// TIA Portal V17 export
// export: Created 2023-02-13T11:16:47.4650946Z, ExportSetting WithDefaults, DisplayName Totally Integrated Automation Portal, DisplayVersion V17, DisplayName TIA Portal Openness, DisplayVersion V17, DisplayName TIA Portal Teamcenter Gateway, DisplayVersion V17, DisplayName TIA Portal Version Control Interface, DisplayVersion V17, DisplayName SINAMICS Startdrive Advanced, DisplayVersion V17, DisplayName SINAMICS Startdrive G130, G150, S120, S150, SINAMICS MV, S210, DisplayVersion V17, DisplayName SINAMICS Startdrive G110M, G120, G120C, G120D, G120P, G115D, DisplayVersion V17, DisplayName STEP 7 Professional, DisplayVersion V17, DisplayName STEP 7 Safety, DisplayVersion V17, DisplayName WinCC Professional, DisplayVersion V17
FUNCTION_BLOCK "Homomix"   // FB18, LAD
{ S7_Optimized_Access := 'TRUE' }
VERSION : 0.1
// stored: AutoNumber true, IsIECCheckEnabled false, IsRetainMemResEnabled false, MemoryReserve 100, SetENOAutomatically false, UDAEnableTagReadback false
   VAR_INPUT
      "Level LL" : Bool;
      IN_FBAV_ProWater : Bool;
      IN_FBAV_HW : Bool;
      IN_FBAV_CIP_Tank : Bool;
      IN_FBAV_CIP_Line : Bool;
      IN_FBAV_Outlet : Bool;
      IN_FBAV_Transfer : Bool;
      IN_FBP_Transfer : Bool;
      IN_FBP_Transfer_SP : Real;
      IN_FBP_CIP : Bool;
      IN_FBP_CIP_SP : Real;
      IN_CIP_Enable : Bool;
      IN_CIP_LineOpen : Bool;
      "CIP Pulse" : Bool;
      "CIP Request OK" : Bool;
      "CIP Supply ON" : Bool;
      "CIP In Progress" : Bool;
      "CIP Complete" : Bool;
      IN_Dose_Run : Bool;
      IN_Dose_Held : Bool;
      IN_Dose_Complete : Bool;
      IN_Dose_Valve_Cmd : Bool;
      IN_Dose_Pump_Cmd : Bool;
      IN_Dose_Pump_Sp : Real;
      IN_Dose_LineOK : Bool;
      "ProWater Ready" : Bool;
      "ProWater En" : Bool;
      "HW Ready" : Bool;
      "HW En" : Bool;
      "CIP Busy" : Bool;
      IN_LDT : Date_And_Time;
   END_VAR
   VAR_OUTPUT
      Out_AV_ProWater : Bool;
      Out_AV_HW : Bool;
      Out_AV_CIP_Tank : Bool;
      Out_AV_CIP_Line : Bool;
      Out_AV_Outlet : Bool;
      Out_AV_Transfer : Bool;
      Out_P_Transfer : Bool;
      Out_P_Transfer_SP : Real;
      Out_P_CIP : Bool;
      Out_P_CIP_SP : Real;
      Out_XA : Bool;
      Out_XA_SP : Real;
      Out_Prod_Ready : Bool;
      Out_Tank_Ready : Bool;
      Out_CIP_Tank_Req : Bool;
      Out_CIP_Line_Req : Bool;
      Out_CIP_LineOpen : Bool;
   END_VAR
   VAR
      Cmd : Struct
         Ready_for_Transfer : Bool;
         "CIP Tank" : Bool;
         "CIP Line" : Bool;
         "Agi Mode" : Bool;
         "Agi ON OFF" : Bool;
      END_STRUCT;
   END_VAR
   VAR RETAIN
      Param : Struct
         "CIP Pump SP" : Real := 50.0;
         "Agi SP" : Real := 50.0;
         Dose_HW_SP : Real;
         Dose_ProWater_SP : Real;
         LastDose_HW : Real;
         LastDose_ProWater : Real;
      END_STRUCT;
   END_VAR
   VAR
      State : Struct
         "Tank LL" : Bool;
         "CIP Tank" : Bool;
         "CIP Tank Ena" : Bool;
         "CIP Line" : Bool;
         "CIP Line Ena" : Bool;
         "CIP Return On" : Bool;
         "Dose EN" : Bool;
         ProWater_Inloading : Bool;
         HW_Inloading : Bool;
         Tank_Inloading : Bool;
         "Ready For Transfer" : Bool;
         "Ready For Transfer EN" : Bool;
         Transfer_On_Prog : Bool;
         "CIP Req" : Bool;
      END_STRUCT;
      Dose : Struct
         Dose_Start : DWord;
         Dose_Pause : DWord;
         Dose_Stop : DWord;
         Dose_State : DWord;
         Dose_Tank_Available : Word;
         Dose_Prod_Ready : Word;
         Dose_Header_Req : DWord;
         Dose_EN : Word;
      END_STRUCT;
      SP_ProWater : "Raw_Pulse";
      SP_HW { S7_SetPoint := 'True'} : "Raw_Pulse";
      Dose_ProWater { S7_SetPoint := 'True'} : "DOSE";
      Dose_HW { S7_SetPoint := 'True'} : "DOSE";
      r : Struct
         PosE1 : Bool;
         PosE2 : Bool;
         PosE3 : Bool;
         PosE4 : Bool;
         PosE5 : Bool;
         PosE6 : Bool;
         PosE7 : Bool;
         PosE8 : Bool;
         PosE9 : Bool;
         PosE10 : Bool;
         PosE11 : Bool;
         PosE12 : Bool;
         PosE13 : Bool;
         PosE14 : Bool;
         PosE15 : Bool;
         PosE16 : Bool;
         PosE17 : Bool;
         PosE18 : Bool;
         PosE19 : Bool;
         PosE20 : Bool;
         PosE21 : Bool;
         PosE22 : Bool;
         PosE23 : Bool;
         PosE24 : Bool;
         PosE25 : Bool;
         PosE26 : Bool;
         PosE27 : Bool;
         PosE28 : Bool;
         PosE29 : Bool;
         PosE30 : Bool;
         PosE31 : Bool;
         PosE32 : Bool;
      END_STRUCT;
      CIPRetOn_Time : TON_TIME;
      CIPRetOff_Time { S7_SetPoint := 'True'} : TON_TIME;
      Actuator : Struct
         AV_Transfer : Bool;
         AV_Outlet : Bool;
         AV_CIP : Bool;
         P_Transfer : Bool;
         P_CIP : Bool;
      END_STRUCT;
      alwaysOn : Bool;
   END_VAR
   VAR RETAIN
      TimerON : Struct
         TimerON_1 : TON_TIME;
         TimerON_2 { S7_SetPoint := 'True'} : TON_TIME;
         TimerON_3 { S7_SetPoint := 'True'} : TON_TIME;
         TimerON_4 { S7_SetPoint := 'True'} : TON_TIME;
         TimerON_5 { S7_SetPoint := 'True'} : TON_TIME;
         TimerON_6 { S7_SetPoint := 'True'} : TON_TIME;
         TimerON_7 { S7_SetPoint := 'True'} : TON_TIME;
         TimerON_8 { S7_SetPoint := 'True'} : TON_TIME;
      END_STRUCT;
   END_VAR
   VAR_TEMP
      b_transfer : Bool;
   END_VAR
   // SP_ProWater.Para."SP_Qty_Fine%" := 10.0;
   // SP_HW.Para."SP_Qty_Fine%" := 10.0;
   // TimerON.TimerON_1.PT := T#10s;
   // TimerON.TimerON_2.PT := T#10s;
   // TimerON.TimerON_3.PT := T#10s;
   // TimerON.TimerON_4.PT := T#10s;
   // TimerON.TimerON_5.PT := T#10s;
   // TimerON.TimerON_6.PT := T#10s;
   // TimerON.TimerON_7.PT := T#10s;
   // TimerON.TimerON_8.PT := T#10s;
   VAR_TEMP   // added for the SCL form of the ladder/FBD networks
      _w1 : Bool;
      _w2 : Bool;
   END_VAR
BEGIN

REGION Network 1: Always ON
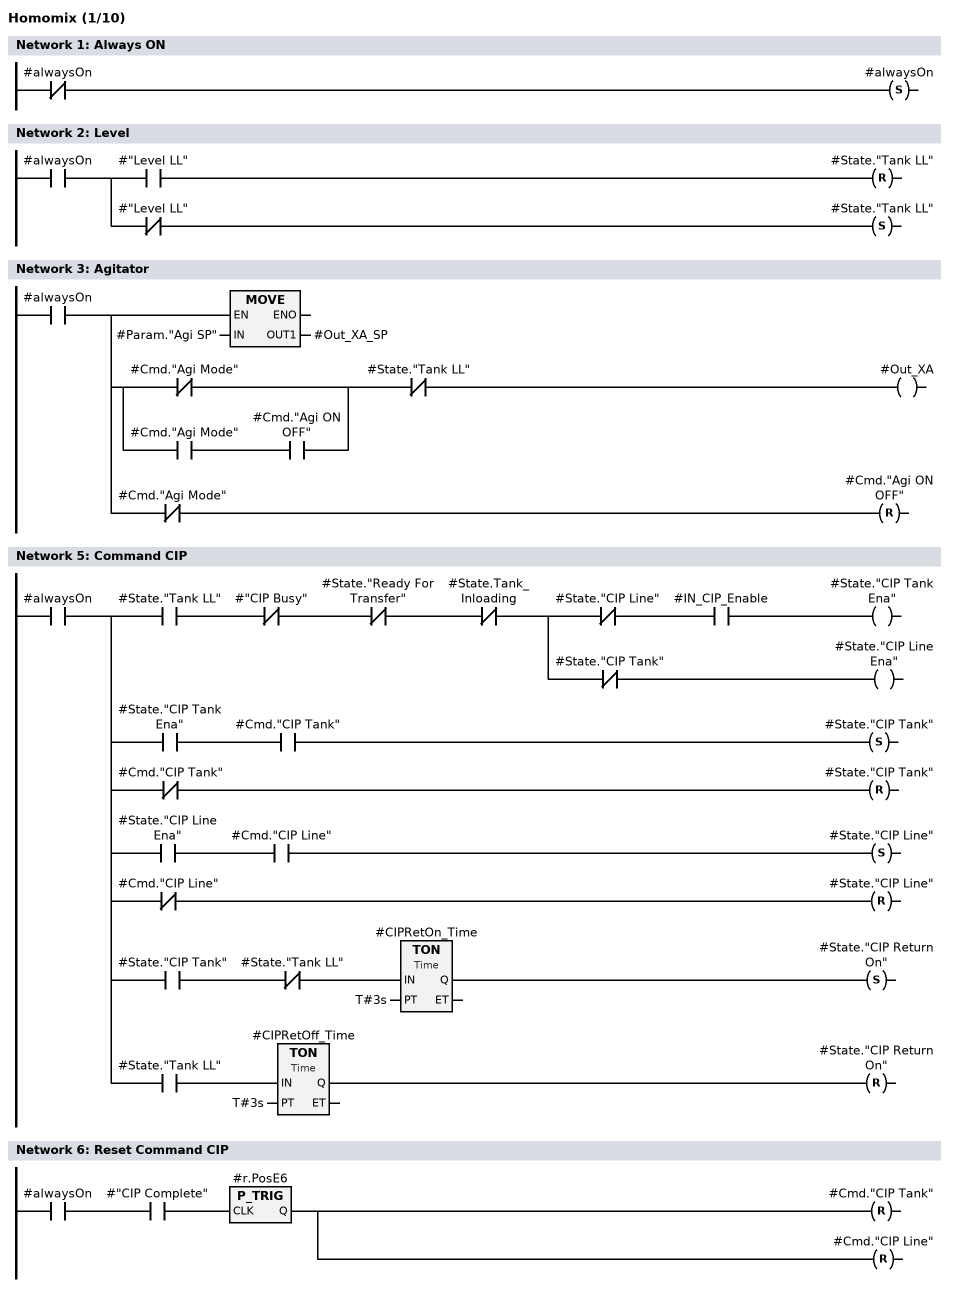
   RUNG wire#powerrail
      I_Contact( #alwaysOn )
      S_Coil( #alwaysOn )
   END_RUNG
   // the same network as SCL:
   IF NOT #alwaysOn THEN #alwaysOn := TRUE; END_IF;
END_REGION

REGION Network 2: Level
   RUNG wire#powerrail
      Contact( #alwaysOn )
      wire#w1
      Contact( #"Level LL" )
      R_Coil( #State."Tank LL" )
   END_RUNG
   RUNG wire#w1
      I_Contact( #"Level LL" )
      S_Coil( #State."Tank LL" )
   END_RUNG
   // the same network as SCL:
   IF #alwaysOn AND #"Level LL" THEN #State."Tank LL" := FALSE; END_IF;
   IF #alwaysOn AND NOT #"Level LL" THEN #State."Tank LL" := TRUE; END_IF;
END_REGION

REGION Network 3: Agitator
   RUNG wire#powerrail
      Contact( #alwaysOn )
      wire#w1
      Move(in := #Param."Agi SP", out1 => #Out_XA_SP)
   END_RUNG
   RUNG wire#w1
      I_Contact( #Cmd."Agi Mode" )
      wire#w2
      I_Contact( #State."Tank LL" )
      Coil( #Out_XA )
   END_RUNG
   RUNG wire#w1
      Contact( #Cmd."Agi Mode" )
      Contact( #Cmd."Agi ON OFF" )
   END_RUNG wire#w2
   RUNG wire#w1
      I_Contact( #Cmd."Agi Mode" )
      R_Coil( #Cmd."Agi ON OFF" )
   END_RUNG
   // the same network as SCL:
   IF #alwaysOn THEN #Out_XA_SP := #Param."Agi SP"; END_IF;
   #Out_XA := #alwaysOn AND (NOT #Cmd."Agi Mode" OR (#Cmd."Agi Mode" AND #Cmd."Agi ON OFF")) AND NOT #State."Tank LL";
   IF #alwaysOn AND NOT #Cmd."Agi Mode" THEN #Cmd."Agi ON OFF" := FALSE; END_IF;
END_REGION

REGION Network 5: Command CIP
   RUNG wire#powerrail
      Contact( #alwaysOn )
      wire#w1
      Contact( #State."Tank LL" )
      I_Contact( #"CIP Busy" )
      I_Contact( #State."Ready For Transfer" )
      I_Contact( #State.Tank_Inloading )
      wire#w2
      I_Contact( #State."CIP Line" )
      Contact( #IN_CIP_Enable )
      Coil( #State."CIP Tank Ena" )
   END_RUNG
   RUNG wire#w2
      I_Contact( #State."CIP Tank" )
      Coil( #State."CIP Line Ena" )
   END_RUNG
   RUNG wire#w1
      Contact( #State."CIP Tank Ena" )
      Contact( #Cmd."CIP Tank" )
      S_Coil( #State."CIP Tank" )
   END_RUNG
   RUNG wire#w1
      I_Contact( #Cmd."CIP Tank" )
      R_Coil( #State."CIP Tank" )
   END_RUNG
   RUNG wire#w1
      Contact( #State."CIP Line Ena" )
      Contact( #Cmd."CIP Line" )
      S_Coil( #State."CIP Line" )
   END_RUNG
   RUNG wire#w1
      I_Contact( #Cmd."CIP Line" )
      R_Coil( #State."CIP Line" )
   END_RUNG
   RUNG wire#w1
      Contact( #State."CIP Tank" )
      I_Contact( #State."Tank LL" )
      { S7_Templates := "time_type := Time" } #CIPRetOn_Time.TON(pt := T#3s, et =>)
      S_Coil( #State."CIP Return On" )
   END_RUNG
   RUNG wire#w1
      Contact( #State."Tank LL" )
      { S7_Templates := "time_type := Time" } #CIPRetOff_Time.TON(pt := T#3s, et =>)
      R_Coil( #State."CIP Return On" )
   END_RUNG
   // the same network as SCL:
   #_w1 := #alwaysOn AND #State."Tank LL" AND NOT #"CIP Busy" AND NOT #State."Ready For Transfer" AND NOT #State.Tank_Inloading;
   #State."CIP Tank Ena" := #_w1 AND NOT #State."CIP Line" AND #IN_CIP_Enable;
   #State."CIP Line Ena" := #_w1 AND NOT #State."CIP Tank";
   IF #alwaysOn AND #State."CIP Tank Ena" AND #Cmd."CIP Tank" THEN #State."CIP Tank" := TRUE; END_IF;
   IF #alwaysOn AND NOT #Cmd."CIP Tank" THEN #State."CIP Tank" := FALSE; END_IF;
   IF #alwaysOn AND #State."CIP Line Ena" AND #Cmd."CIP Line" THEN #State."CIP Line" := TRUE; END_IF;
   IF #alwaysOn AND NOT #Cmd."CIP Line" THEN #State."CIP Line" := FALSE; END_IF;
   #CIPRetOn_Time(IN := #alwaysOn AND #State."CIP Tank" AND NOT #State."Tank LL", PT := T#3s);   // TON
   IF #CIPRetOn_Time.Q THEN #State."CIP Return On" := TRUE; END_IF;
   #CIPRetOff_Time(IN := #alwaysOn AND #State."Tank LL", PT := T#3s);   // TON
   IF #CIPRetOff_Time.Q THEN #State."CIP Return On" := FALSE; END_IF;
END_REGION

REGION Network 6: Reset Command CIP
   RUNG wire#powerrail
      Contact( #alwaysOn )
      Contact( #"CIP Complete" )
      P_Trig( #r.PosE6 )
      wire#w1
      R_Coil( #Cmd."CIP Tank" )
   END_RUNG
   RUNG wire#w1
      R_Coil( #Cmd."CIP Line" )
   END_RUNG
   // the same network as SCL:
   #_w1 := #alwaysOn AND #"CIP Complete";
   #_w2 := #_w1 AND NOT #r.PosE6;   // rising edge
   #r.PosE6 := #_w1;
   IF #_w2 THEN
       #Cmd."CIP Tank" := FALSE;
       #Cmd."CIP Line" := FALSE;
   END_IF;
END_REGION

REGION Network 7: CIP Request and CIP Line Open
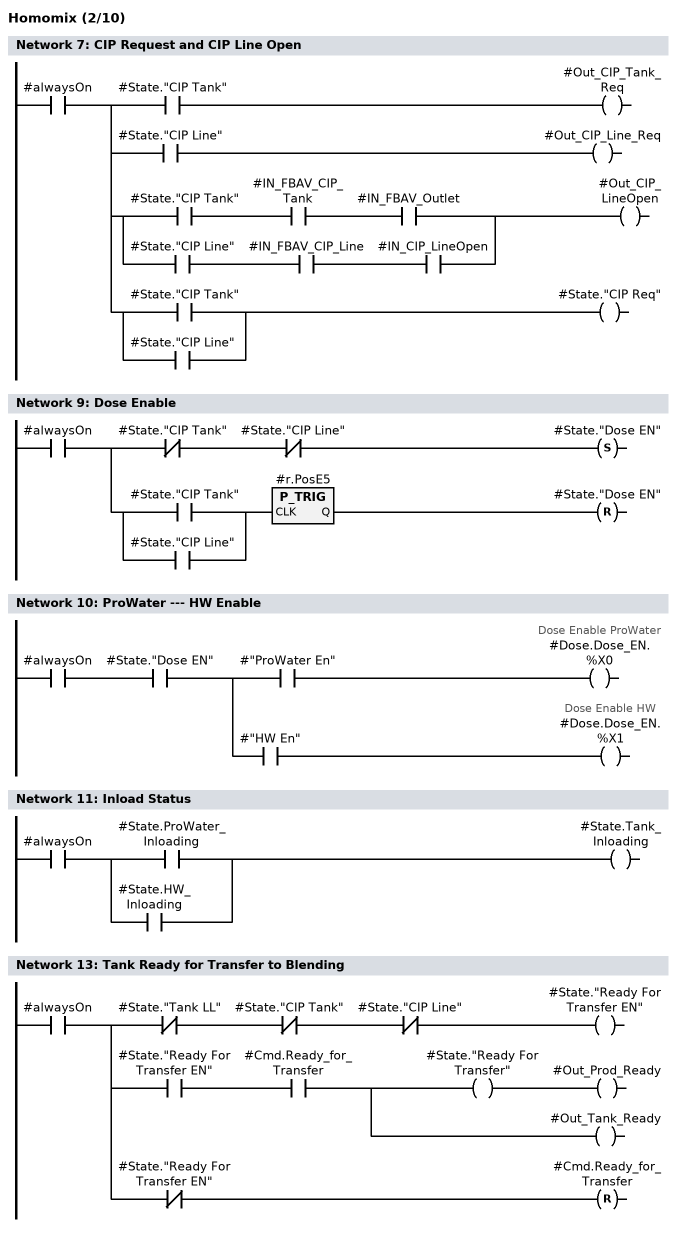
   RUNG wire#powerrail
      Contact( #alwaysOn )
      wire#w1
      Contact( #State."CIP Tank" )
      Coil( #Out_CIP_Tank_Req )
   END_RUNG
   RUNG wire#w1
      Contact( #State."CIP Line" )
      Coil( #Out_CIP_Line_Req )
   END_RUNG
   RUNG wire#w1
      Contact( #State."CIP Tank" )
      Contact( #IN_FBAV_CIP_Tank )
      Contact( #IN_FBAV_Outlet )
      wire#w2
      Coil( #Out_CIP_LineOpen )
   END_RUNG
   RUNG wire#w1
      Contact( #State."CIP Line" )
      Contact( #IN_FBAV_CIP_Line )
      Contact( #IN_CIP_LineOpen )
   END_RUNG wire#w2
   RUNG wire#w1
      Contact( #State."CIP Tank" )
      wire#w3
      Coil( #State."CIP Req" )
   END_RUNG
   RUNG wire#w1
      Contact( #State."CIP Line" )
   END_RUNG wire#w3
   // the same network as SCL:
   #Out_CIP_Tank_Req := #alwaysOn AND #State."CIP Tank";
   #Out_CIP_Line_Req := #alwaysOn AND #State."CIP Line";
   #Out_CIP_LineOpen := #alwaysOn AND ((#State."CIP Tank" AND #IN_FBAV_CIP_Tank AND #IN_FBAV_Outlet) OR (#State."CIP Line" AND #IN_FBAV_CIP_Line AND #IN_CIP_LineOpen));
   #State."CIP Req" := #alwaysOn AND (#State."CIP Tank" OR #State."CIP Line");
END_REGION

REGION Network 9: Dose Enable
   RUNG wire#powerrail
      Contact( #alwaysOn )
      wire#w1
      I_Contact( #State."CIP Tank" )
      I_Contact( #State."CIP Line" )
      S_Coil( #State."Dose EN" )
   END_RUNG
   RUNG wire#w1
      Contact( #State."CIP Tank" )
      wire#w2
      P_Trig( #r.PosE5 )
      R_Coil( #State."Dose EN" )
   END_RUNG
   RUNG wire#w1
      Contact( #State."CIP Line" )
   END_RUNG wire#w2
   // the same network as SCL:
   IF #alwaysOn AND NOT #State."CIP Tank" AND NOT #State."CIP Line" THEN #State."Dose EN" := TRUE; END_IF;
   #_w1 := #alwaysOn AND (#State."CIP Tank" OR #State."CIP Line");
   #_w2 := #_w1 AND NOT #r.PosE5;   // rising edge
   #r.PosE5 := #_w1;
   IF #_w2 THEN #State."Dose EN" := FALSE; END_IF;
END_REGION

REGION Network 10: ProWater --- HW Enable
   RUNG wire#powerrail
      Contact( #alwaysOn )
      Contact( #State."Dose EN" )
      wire#w1
      Contact( #"ProWater En" )
      Coil( #Dose.Dose_EN.%X0 )   // Dose Enable ProWater
   END_RUNG
   RUNG wire#w1
      Contact( #"HW En" )
      Coil( #Dose.Dose_EN.%X1 )   // Dose Enable HW
   END_RUNG
   // the same network as SCL:
   #_w1 := #alwaysOn AND #State."Dose EN";
   #Dose.Dose_EN.%X0 := #_w1 AND #"ProWater En";   // Dose Enable ProWater
   #Dose.Dose_EN.%X1 := #_w1 AND #"HW En";   // Dose Enable HW
END_REGION

REGION Network 11: Inload Status
   RUNG wire#powerrail
      Contact( #alwaysOn )
      wire#w1
      Contact( #State.ProWater_Inloading )
      wire#w2
      Coil( #State.Tank_Inloading )
   END_RUNG
   RUNG wire#w1
      Contact( #State.HW_Inloading )
   END_RUNG wire#w2
   // the same network as SCL:
   #State.Tank_Inloading := #alwaysOn AND (#State.ProWater_Inloading OR #State.HW_Inloading);
END_REGION

REGION Network 13: Tank Ready for Transfer to Blending
   RUNG wire#powerrail
      Contact( #alwaysOn )
      wire#w1
      I_Contact( #State."Tank LL" )
      I_Contact( #State."CIP Tank" )
      I_Contact( #State."CIP Line" )
      Coil( #State."Ready For Transfer EN" )
   END_RUNG
   RUNG wire#w1
      Contact( #State."Ready For Transfer EN" )
      Contact( #Cmd.Ready_for_Transfer )
      wire#w2
      Coil( #State."Ready For Transfer" )
      Coil( #Out_Prod_Ready )
   END_RUNG
   RUNG wire#w2
      Coil( #Out_Tank_Ready )
   END_RUNG
   RUNG wire#w1
      I_Contact( #State."Ready For Transfer EN" )
      R_Coil( #Cmd.Ready_for_Transfer )
   END_RUNG
   // the same network as SCL:
   #State."Ready For Transfer EN" := #alwaysOn AND NOT #State."Tank LL" AND NOT #State."CIP Tank" AND NOT #State."CIP Line";
   #State."Ready For Transfer" := #alwaysOn AND #State."Ready For Transfer EN" AND #Cmd.Ready_for_Transfer;
   #Out_Prod_Ready := #State."Ready For Transfer";
   #Out_Tank_Ready := #State."Ready For Transfer";
   IF #alwaysOn AND NOT #State."Ready For Transfer EN" THEN #Cmd.Ready_for_Transfer := FALSE; END_IF;
END_REGION

REGION Network 14: Transfer to Blending AV and Pump
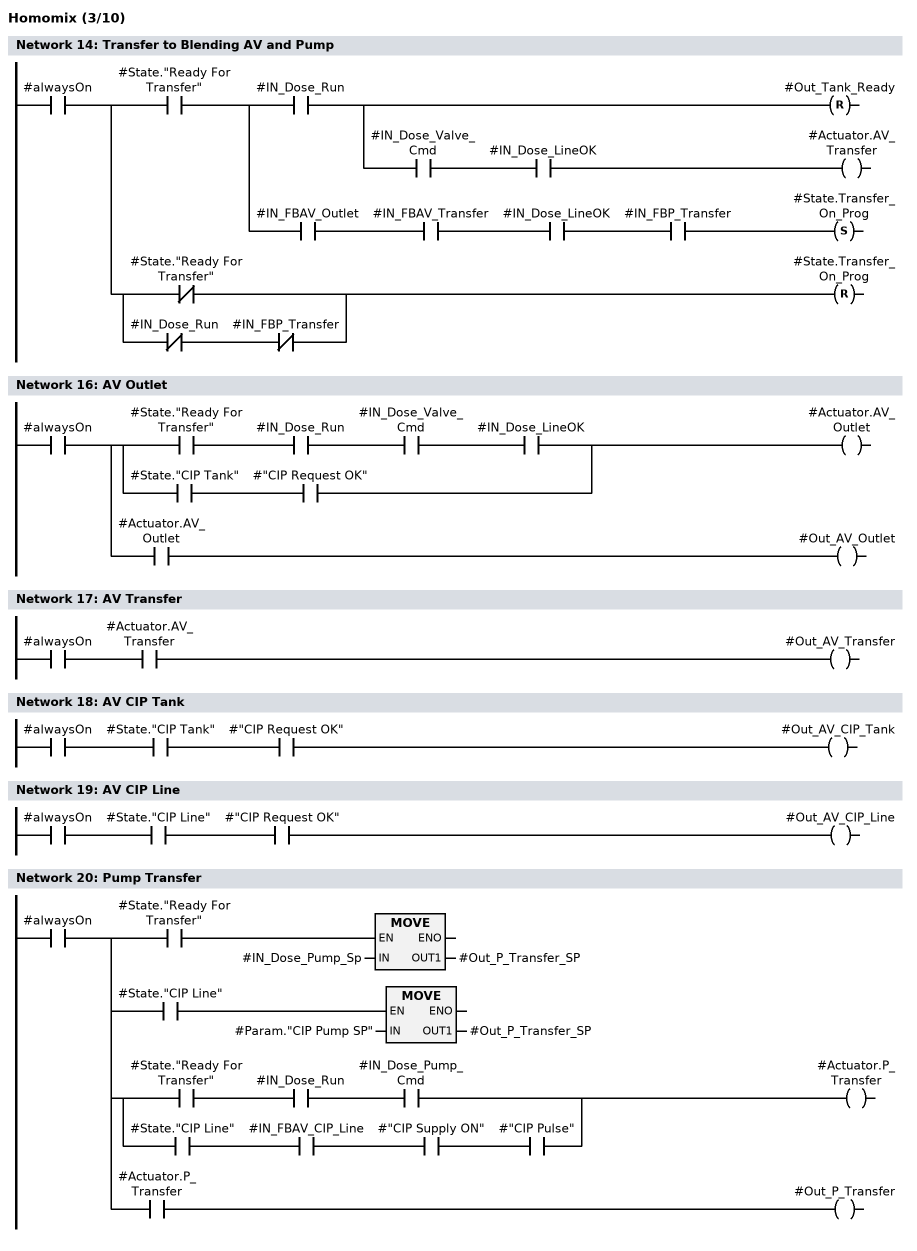
   RUNG wire#powerrail
      Contact( #alwaysOn )
      wire#w1
      Contact( #State."Ready For Transfer" )
      wire#w2
      Contact( #IN_Dose_Run )
      wire#w3
      R_Coil( #Out_Tank_Ready )
   END_RUNG
   RUNG wire#w3
      Contact( #IN_Dose_Valve_Cmd )
      Contact( #IN_Dose_LineOK )
      Coil( #Actuator.AV_Transfer )
   END_RUNG
   RUNG wire#w2
      Contact( #IN_FBAV_Outlet )
      Contact( #IN_FBAV_Transfer )
      Contact( #IN_Dose_LineOK )
      Contact( #IN_FBP_Transfer )
      S_Coil( #State.Transfer_On_Prog )
   END_RUNG
   RUNG wire#w1
      I_Contact( #State."Ready For Transfer" )
      wire#w4
      R_Coil( #State.Transfer_On_Prog )
   END_RUNG
   RUNG wire#w1
      I_Contact( #IN_Dose_Run )
      I_Contact( #IN_FBP_Transfer )
   END_RUNG wire#w4
   // the same network as SCL:
   #_w1 := #alwaysOn AND #State."Ready For Transfer";
   #_w2 := #_w1 AND #IN_Dose_Run;
   IF #_w2 THEN #Out_Tank_Ready := FALSE; END_IF;
   #Actuator.AV_Transfer := #_w2 AND #IN_Dose_Valve_Cmd AND #IN_Dose_LineOK;
   IF #_w1 AND #IN_FBAV_Outlet AND #IN_FBAV_Transfer AND #IN_Dose_LineOK AND #IN_FBP_Transfer THEN
       #State.Transfer_On_Prog := TRUE;
   END_IF;
   IF #alwaysOn AND (NOT #State."Ready For Transfer" OR (NOT #IN_Dose_Run AND NOT #IN_FBP_Transfer)) THEN
       #State.Transfer_On_Prog := FALSE;
   END_IF;
END_REGION

REGION Network 16: AV Outlet
   RUNG wire#powerrail
      Contact( #alwaysOn )
      wire#w1
      Contact( #State."Ready For Transfer" )
      Contact( #IN_Dose_Run )
      Contact( #IN_Dose_Valve_Cmd )
      Contact( #IN_Dose_LineOK )
      wire#w2
      Coil( #Actuator.AV_Outlet )
   END_RUNG
   RUNG wire#w1
      Contact( #State."CIP Tank" )
      Contact( #"CIP Request OK" )
   END_RUNG wire#w2
   RUNG wire#w1
      Contact( #Actuator.AV_Outlet )
      Coil( #Out_AV_Outlet )
   END_RUNG
   // the same network as SCL:
   #Actuator.AV_Outlet := #alwaysOn AND ((#State."Ready For Transfer" AND #IN_Dose_Run AND #IN_Dose_Valve_Cmd AND #IN_Dose_LineOK) OR (#State."CIP Tank" AND #"CIP Request OK"));
   #Out_AV_Outlet := #alwaysOn AND #Actuator.AV_Outlet;
END_REGION

REGION Network 17: AV Transfer
   RUNG wire#powerrail
      Contact( #alwaysOn )
      Contact( #Actuator.AV_Transfer )
      Coil( #Out_AV_Transfer )
   END_RUNG
   // the same network as SCL:
   #Out_AV_Transfer := #alwaysOn AND #Actuator.AV_Transfer;
END_REGION

REGION Network 18: AV CIP Tank
   RUNG wire#powerrail
      Contact( #alwaysOn )
      Contact( #State."CIP Tank" )
      Contact( #"CIP Request OK" )
      Coil( #Out_AV_CIP_Tank )
   END_RUNG
   // the same network as SCL:
   #Out_AV_CIP_Tank := #alwaysOn AND #State."CIP Tank" AND #"CIP Request OK";
END_REGION

REGION Network 19: AV CIP Line
   RUNG wire#powerrail
      Contact( #alwaysOn )
      Contact( #State."CIP Line" )
      Contact( #"CIP Request OK" )
      Coil( #Out_AV_CIP_Line )
   END_RUNG
   // the same network as SCL:
   #Out_AV_CIP_Line := #alwaysOn AND #State."CIP Line" AND #"CIP Request OK";
END_REGION

REGION Network 20: Pump Transfer
   RUNG wire#powerrail
      Contact( #alwaysOn )
      wire#w1
      Contact( #State."Ready For Transfer" )
      Move(in := #IN_Dose_Pump_Sp, out1 => #Out_P_Transfer_SP)
   END_RUNG
   RUNG wire#w1
      Contact( #State."CIP Line" )
      Move(in := #Param."CIP Pump SP", out1 => #Out_P_Transfer_SP)
   END_RUNG
   RUNG wire#w1
      Contact( #State."Ready For Transfer" )
      Contact( #IN_Dose_Run )
      Contact( #IN_Dose_Pump_Cmd )
      wire#w2
      Coil( #Actuator.P_Transfer )
   END_RUNG
   RUNG wire#w1
      Contact( #State."CIP Line" )
      Contact( #IN_FBAV_CIP_Line )
      Contact( #"CIP Supply ON" )
      Contact( #"CIP Pulse" )
   END_RUNG wire#w2
   RUNG wire#w1
      Contact( #Actuator.P_Transfer )
      Coil( #Out_P_Transfer )
   END_RUNG
   // the same network as SCL:
   IF #alwaysOn AND #State."Ready For Transfer" THEN #Out_P_Transfer_SP := #IN_Dose_Pump_Sp; END_IF;
   IF #alwaysOn AND #State."CIP Line" THEN #Out_P_Transfer_SP := #Param."CIP Pump SP"; END_IF;
   #Actuator.P_Transfer := #alwaysOn AND ((#State."Ready For Transfer" AND #IN_Dose_Run AND #IN_Dose_Pump_Cmd) OR (#State."CIP Line" AND #IN_FBAV_CIP_Line AND #"CIP Supply ON" AND #"CIP Pulse"));
   #Out_P_Transfer := #alwaysOn AND #Actuator.P_Transfer;
END_REGION

REGION Network 21: Pump CIP Tank
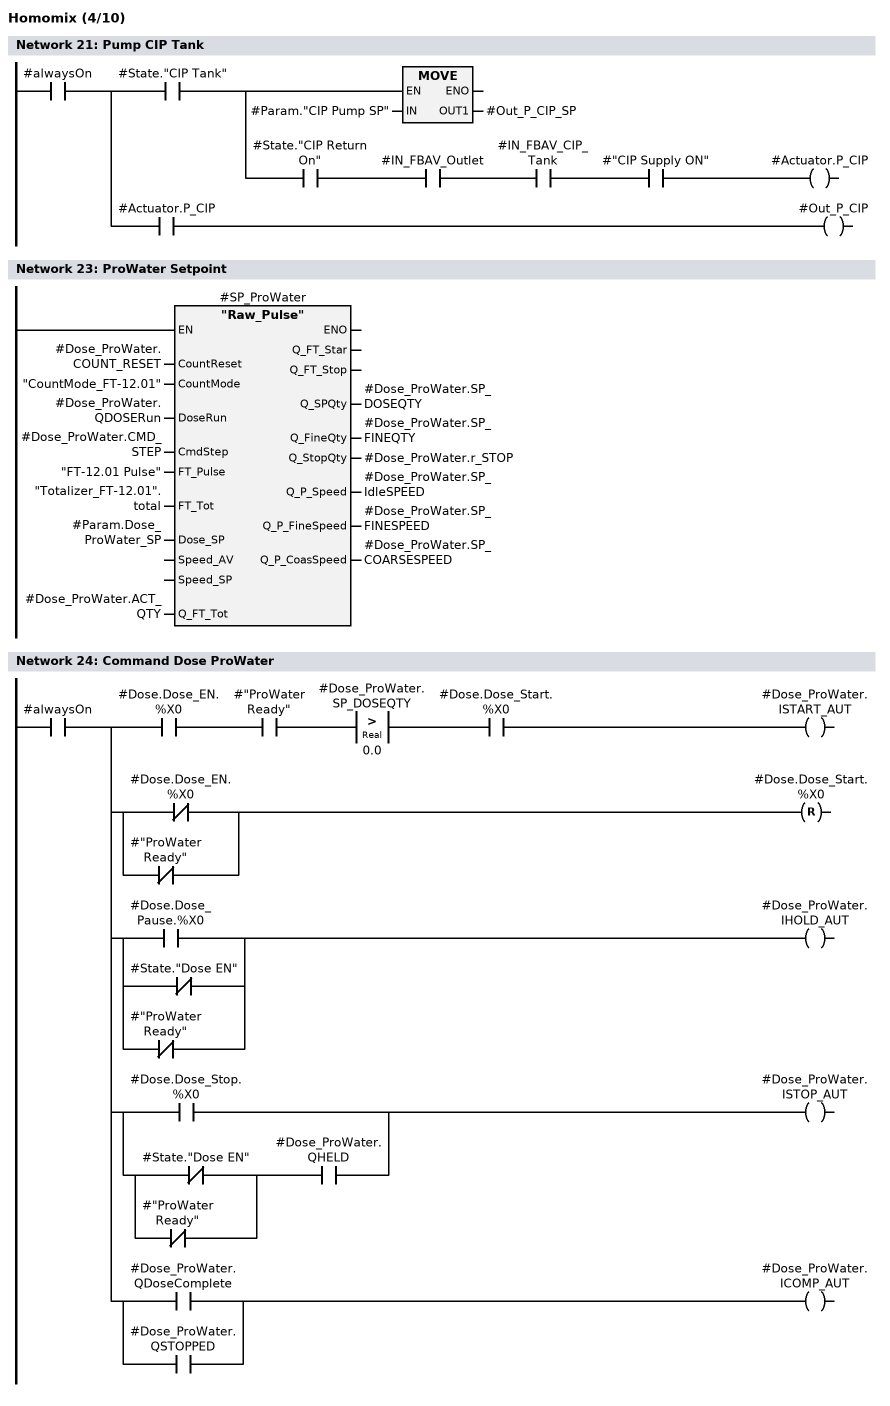
   RUNG wire#powerrail
      Contact( #alwaysOn )
      wire#w1
      Contact( #State."CIP Tank" )
      wire#w2
      Move(in := #Param."CIP Pump SP", out1 => #Out_P_CIP_SP)
   END_RUNG
   RUNG wire#w2
      Contact( #State."CIP Return On" )
      Contact( #IN_FBAV_Outlet )
      Contact( #IN_FBAV_CIP_Tank )
      Contact( #"CIP Supply ON" )
      Coil( #Actuator.P_CIP )
   END_RUNG
   RUNG wire#w1
      Contact( #Actuator.P_CIP )
      Coil( #Out_P_CIP )
   END_RUNG
   // the same network as SCL:
   #_w1 := #alwaysOn AND #State."CIP Tank";
   IF #_w1 THEN #Out_P_CIP_SP := #Param."CIP Pump SP"; END_IF;
   #Actuator.P_CIP := #_w1 AND #State."CIP Return On" AND #IN_FBAV_Outlet AND #IN_FBAV_CIP_Tank AND #"CIP Supply ON";
   #Out_P_CIP := #alwaysOn AND #Actuator.P_CIP;
END_REGION

REGION Network 23: ProWater Setpoint
   RUNG wire#powerrail
      #SP_ProWater(CountReset := #Dose_ProWater.COUNT_RESET, CountMode := "CountMode_FT-12.01", DoseRun := #Dose_ProWater.QDOSERun, CmdStep := #Dose_ProWater.CMD_STEP, FT_Pulse := "FT-12.01 Pulse", FT_Tot := "Totalizer_FT-12.01".total, Dose_SP := #Param.Dose_ProWater_SP, Speed_AV :=, Speed_SP :=, Q_FT_Tot := #Dose_ProWater.ACT_QTY, Q_FT_Star =>, Q_FT_Stop =>, Q_SPQty => #Dose_ProWater.SP_DOSEQTY, Q_FineQty => #Dose_ProWater.SP_FINEQTY, Q_StopQty => #Dose_ProWater.r_STOP, Q_P_Speed => #Dose_ProWater.SP_IdleSPEED, Q_P_FineSpeed => #Dose_ProWater.SP_FINESPEED, Q_P_CoasSpeed => #Dose_ProWater.SP_COARSESPEED)
   END_RUNG
   // the same network as SCL:
   #SP_ProWater(CountReset := #Dose_ProWater.COUNT_RESET,   // "Raw_Pulse"
                CountMode := "CountMode_FT-12.01",
                DoseRun := #Dose_ProWater.QDOSERun,
                CmdStep := #Dose_ProWater.CMD_STEP,
                FT_Pulse := "FT-12.01 Pulse",
                FT_Tot := "Totalizer_FT-12.01".total,
                Dose_SP := #Param.Dose_ProWater_SP,
                Q_FT_Tot := #Dose_ProWater.ACT_QTY,
                Q_SPQty => #Dose_ProWater.SP_DOSEQTY,
                Q_FineQty => #Dose_ProWater.SP_FINEQTY,
                Q_StopQty => #Dose_ProWater.r_STOP,
                Q_P_Speed => #Dose_ProWater.SP_IdleSPEED,
                Q_P_FineSpeed => #Dose_ProWater.SP_FINESPEED,
                Q_P_CoasSpeed => #Dose_ProWater.SP_COARSESPEED);
END_REGION

REGION Network 24: Command Dose ProWater
   RUNG wire#powerrail
      Contact( #alwaysOn )
      wire#w1
      Contact( #Dose.Dose_EN.%X0 )
      Contact( #"ProWater Ready" )
      { S7_Templates := "SrcType := Real" } GT_Contact(in1 := #Dose_ProWater.SP_DOSEQTY, in2 := 0.0)
      Contact( #Dose.Dose_Start.%X0 )
      Coil( #Dose_ProWater.ISTART_AUT )
   END_RUNG
   RUNG wire#w1
      I_Contact( #Dose.Dose_EN.%X0 )
      wire#w2
      R_Coil( #Dose.Dose_Start.%X0 )
   END_RUNG
   RUNG wire#w1
      I_Contact( #"ProWater Ready" )
   END_RUNG wire#w2
   RUNG wire#w1
      Contact( #Dose.Dose_Pause.%X0 )
      wire#w3
      Coil( #Dose_ProWater.IHOLD_AUT )
   END_RUNG
   RUNG wire#w1
      I_Contact( #State."Dose EN" )
   END_RUNG wire#w3
   RUNG wire#w1
      I_Contact( #"ProWater Ready" )
   END_RUNG wire#w3
   RUNG wire#w1
      Contact( #Dose.Dose_Stop.%X0 )
      wire#w4
      Coil( #Dose_ProWater.ISTOP_AUT )
   END_RUNG
   RUNG wire#w1
      I_Contact( #State."Dose EN" )
      wire#w5
      Contact( #Dose_ProWater.QHELD )
   END_RUNG wire#w4
   RUNG wire#w1
      I_Contact( #"ProWater Ready" )
   END_RUNG wire#w5
   RUNG wire#w1
      Contact( #Dose_ProWater.QDoseComplete )
      wire#w6
      Coil( #Dose_ProWater.ICOMP_AUT )
   END_RUNG
   RUNG wire#w1
      Contact( #Dose_ProWater.QSTOPPED )
   END_RUNG wire#w6
   // the same network as SCL:
   #Dose_ProWater.ISTART_AUT := #alwaysOn AND #Dose.Dose_EN.%X0 AND #"ProWater Ready" AND (#Dose_ProWater.SP_DOSEQTY > 0.0) AND #Dose.Dose_Start.%X0;
   IF #alwaysOn AND (NOT #Dose.Dose_EN.%X0 OR NOT #"ProWater Ready") THEN
       #Dose.Dose_Start.%X0 := FALSE;
   END_IF;
   #Dose_ProWater.IHOLD_AUT := #alwaysOn AND (#Dose.Dose_Pause.%X0 OR NOT #State."Dose EN" OR NOT #"ProWater Ready");
   #Dose_ProWater.ISTOP_AUT := #alwaysOn AND (#Dose.Dose_Stop.%X0 OR ((NOT #State."Dose EN" OR NOT #"ProWater Ready") AND #Dose_ProWater.QHELD));
   #Dose_ProWater.ICOMP_AUT := #alwaysOn AND (#Dose_ProWater.QDoseComplete OR #Dose_ProWater.QSTOPPED);
END_REGION

REGION Network 25: Dose ProWater
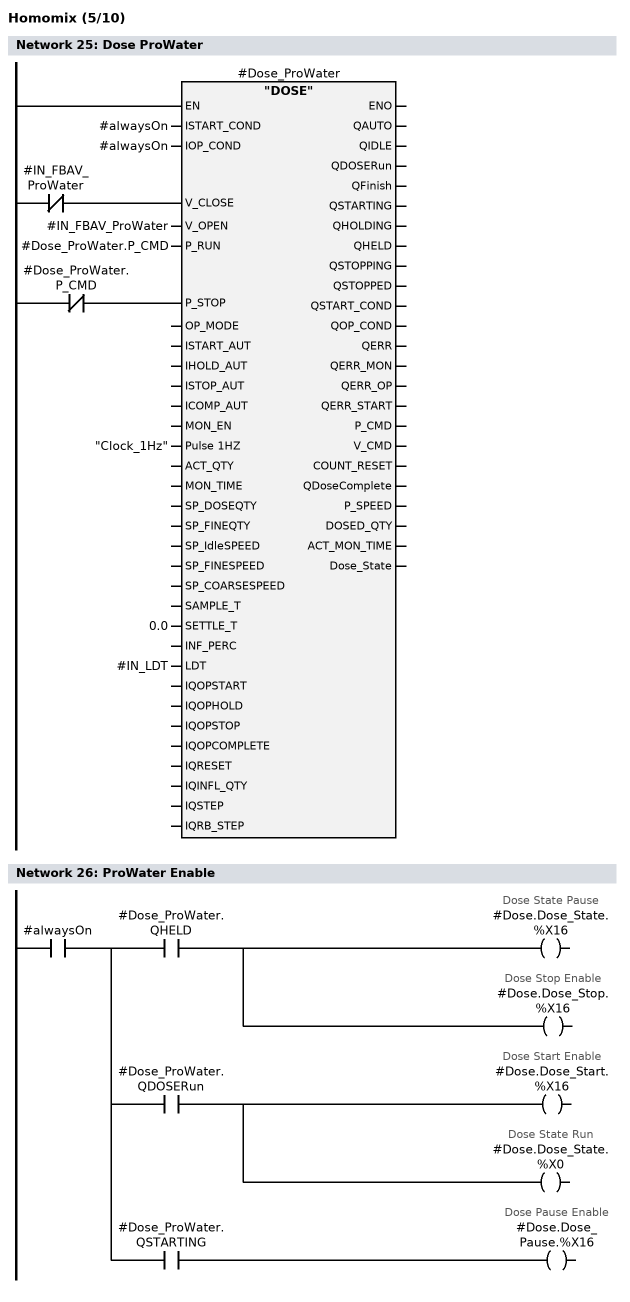
   RUNG wire#powerrail
      #Dose_ProWater(V_CLOSE := wire#w1, P_STOP := wire#w2, ISTART_COND := #alwaysOn, IOP_COND := #alwaysOn, V_OPEN := #IN_FBAV_ProWater, P_RUN := #Dose_ProWater.P_CMD, OP_MODE :=, ISTART_AUT :=, IHOLD_AUT :=, ISTOP_AUT :=, ICOMP_AUT :=, MON_EN :=, "Pulse 1HZ" := "Clock_1Hz", ACT_QTY :=, MON_TIME :=, SP_DOSEQTY :=, SP_FINEQTY :=, SP_IdleSPEED :=, SP_FINESPEED :=, SP_COARSESPEED :=, SAMPLE_T :=, SETTLE_T := 0.0, INF_PERC :=, LDT := #IN_LDT, IQOPSTART :=, IQOPHOLD :=, IQOPSTOP :=, IQOPCOMPLETE :=, IQRESET :=, IQINFL_QTY :=, IQSTEP :=, IQRB_STEP :=, QAUTO =>, QIDLE =>, QDOSERun =>, QFinish =>, QSTARTING =>, QHOLDING =>, QHELD =>, QSTOPPING =>, QSTOPPED =>, QSTART_COND =>, QOP_COND =>, QERR =>, QERR_MON =>, QERR_OP =>, QERR_START =>, P_CMD =>, V_CMD =>, COUNT_RESET =>, QDoseComplete =>, P_SPEED =>, DOSED_QTY =>, ACT_MON_TIME =>, Dose_State =>)
   END_RUNG
   RUNG wire#powerrail
      I_Contact( #IN_FBAV_ProWater )
   END_RUNG wire#w1
   RUNG wire#powerrail
      I_Contact( #Dose_ProWater.P_CMD )
   END_RUNG wire#w2
   // the same network as SCL:
   #Dose_ProWater(ISTART_COND := #alwaysOn,   // "DOSE"
                  IOP_COND := #alwaysOn,
                  V_CLOSE := NOT #IN_FBAV_ProWater,
                  V_OPEN := #IN_FBAV_ProWater,
                  P_RUN := #Dose_ProWater.P_CMD,
                  P_STOP := NOT #Dose_ProWater.P_CMD,
                  "Pulse 1HZ" := "Clock_1Hz",
                  SETTLE_T := 0.0,
                  LDT := #IN_LDT);
END_REGION

REGION Network 26: ProWater Enable
   RUNG wire#powerrail
      Contact( #alwaysOn )
      wire#w1
      Contact( #Dose_ProWater.QHELD )
      wire#w2
      Coil( #Dose.Dose_State.%X16 )   // Dose State Pause
   END_RUNG
   RUNG wire#w2
      Coil( #Dose.Dose_Stop.%X16 )   // Dose Stop Enable
   END_RUNG
   RUNG wire#w1
      Contact( #Dose_ProWater.QDOSERun )
      wire#w3
      Coil( #Dose.Dose_Start.%X16 )   // Dose Start Enable
   END_RUNG
   RUNG wire#w3
      Coil( #Dose.Dose_State.%X0 )   // Dose State Run
   END_RUNG
   RUNG wire#w1
      Contact( #Dose_ProWater.QSTARTING )
      Coil( #Dose.Dose_Pause.%X16 )   // Dose Pause Enable
   END_RUNG
   // the same network as SCL:
   #Dose.Dose_State.%X16 := #alwaysOn AND #Dose_ProWater.QHELD;   // Dose State Pause
   #Dose.Dose_Stop.%X16 := #Dose.Dose_State.%X16;   // Dose Stop Enable
   #Dose.Dose_Start.%X16 := #alwaysOn AND #Dose_ProWater.QDOSERun;   // Dose Start Enable
   #Dose.Dose_State.%X0 := #Dose.Dose_Start.%X16;   // Dose State Run
   #Dose.Dose_Pause.%X16 := #alwaysOn AND #Dose_ProWater.QSTARTING;   // Dose Pause Enable
END_REGION

REGION Network 27: ProWater Header Req and Valve
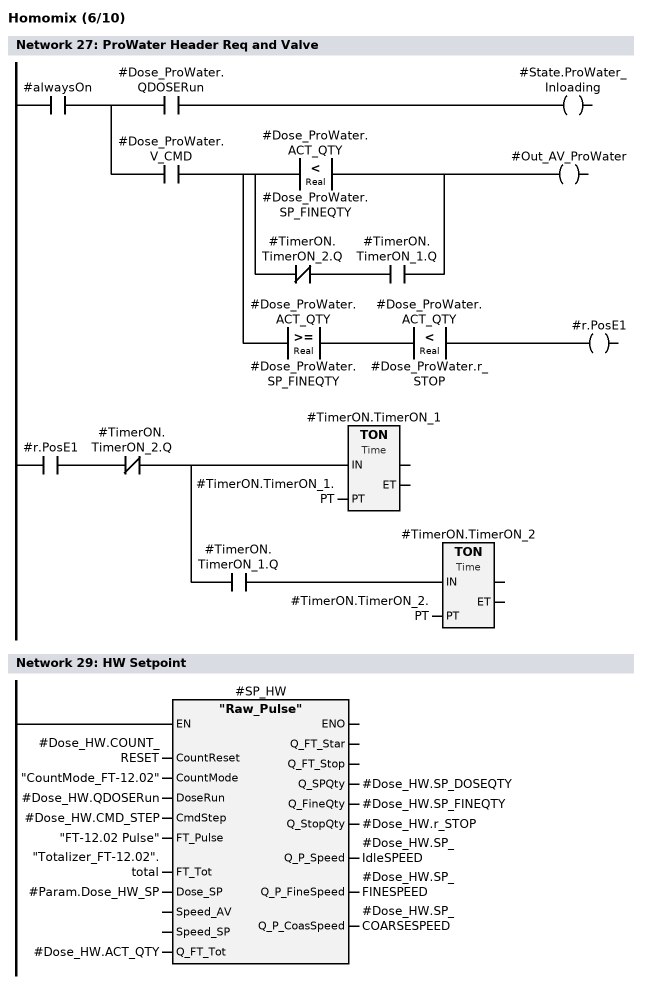
   RUNG wire#powerrail
      Contact( #alwaysOn )
      wire#w1
      Contact( #Dose_ProWater.QDOSERun )
      Coil( #State.ProWater_Inloading )
   END_RUNG
   RUNG wire#w1
      Contact( #Dose_ProWater.V_CMD )
      wire#w2
      { S7_Templates := "SrcType := Real" } LT_Contact(in1 := #Dose_ProWater.ACT_QTY, in2 := #Dose_ProWater.SP_FINEQTY)
      wire#w3
      Coil( #Out_AV_ProWater )
   END_RUNG
   RUNG wire#w2
      I_Contact( #TimerON.TimerON_2.Q )
      Contact( #TimerON.TimerON_1.Q )
   END_RUNG wire#w3
   RUNG wire#w2
      { S7_Templates := "SrcType := Real" } GE_Contact(in1 := #Dose_ProWater.ACT_QTY, in2 := #Dose_ProWater.SP_FINEQTY)
      { S7_Templates := "SrcType := Real" } LT_Contact(in1 := #Dose_ProWater.ACT_QTY, in2 := #Dose_ProWater.r_STOP)
      Coil( #r.PosE1 )
   END_RUNG
   RUNG wire#powerrail
      Contact( #r.PosE1 )
      I_Contact( #TimerON.TimerON_2.Q )
      wire#w4
      { S7_Templates := "time_type := Time" } #TimerON.TimerON_1.TON(pt := #TimerON.TimerON_1.PT, et =>)
   END_RUNG
   RUNG wire#w4
      Contact( #TimerON.TimerON_1.Q )
      { S7_Templates := "time_type := Time" } #TimerON.TimerON_2.TON(pt := #TimerON.TimerON_2.PT, et =>)
   END_RUNG
   // the same network as SCL:
   #State.ProWater_Inloading := #alwaysOn AND #Dose_ProWater.QDOSERun;
   #_w1 := #alwaysOn AND #Dose_ProWater.V_CMD;
   #Out_AV_ProWater := #_w1 AND ((#Dose_ProWater.ACT_QTY < #Dose_ProWater.SP_FINEQTY) OR (NOT #TimerON.TimerON_2.Q AND #TimerON.TimerON_1.Q));
   #r.PosE1 := #_w1 AND (#Dose_ProWater.ACT_QTY >= #Dose_ProWater.SP_FINEQTY) AND (#Dose_ProWater.ACT_QTY < #Dose_ProWater.r_STOP);
   #_w2 := #r.PosE1 AND NOT #TimerON.TimerON_2.Q;
   #TimerON.TimerON_1.TON(IN := #_w2, PT := #TimerON.TimerON_1.PT);
   #TimerON.TimerON_2.TON(IN := #_w2 AND #TimerON.TimerON_1.Q, PT := #TimerON.TimerON_2.PT);
END_REGION

REGION Network 29: HW Setpoint
   RUNG wire#powerrail
      #SP_HW(CountReset := #Dose_HW.COUNT_RESET, CountMode := "CountMode_FT-12.02", DoseRun := #Dose_HW.QDOSERun, CmdStep := #Dose_HW.CMD_STEP, FT_Pulse := "FT-12.02 Pulse", FT_Tot := "Totalizer_FT-12.02".total, Dose_SP := #Param.Dose_HW_SP, Speed_AV :=, Speed_SP :=, Q_FT_Tot := #Dose_HW.ACT_QTY, Q_FT_Star =>, Q_FT_Stop =>, Q_SPQty => #Dose_HW.SP_DOSEQTY, Q_FineQty => #Dose_HW.SP_FINEQTY, Q_StopQty => #Dose_HW.r_STOP, Q_P_Speed => #Dose_HW.SP_IdleSPEED, Q_P_FineSpeed => #Dose_HW.SP_FINESPEED, Q_P_CoasSpeed => #Dose_HW.SP_COARSESPEED)
   END_RUNG
   // the same network as SCL:
   #SP_HW(CountReset := #Dose_HW.COUNT_RESET,   // "Raw_Pulse"
          CountMode := "CountMode_FT-12.02",
          DoseRun := #Dose_HW.QDOSERun,
          CmdStep := #Dose_HW.CMD_STEP,
          FT_Pulse := "FT-12.02 Pulse",
          FT_Tot := "Totalizer_FT-12.02".total,
          Dose_SP := #Param.Dose_HW_SP,
          Q_FT_Tot := #Dose_HW.ACT_QTY,
          Q_SPQty => #Dose_HW.SP_DOSEQTY,
          Q_FineQty => #Dose_HW.SP_FINEQTY,
          Q_StopQty => #Dose_HW.r_STOP,
          Q_P_Speed => #Dose_HW.SP_IdleSPEED,
          Q_P_FineSpeed => #Dose_HW.SP_FINESPEED,
          Q_P_CoasSpeed => #Dose_HW.SP_COARSESPEED);
END_REGION

REGION Network 30: Command Dose HW
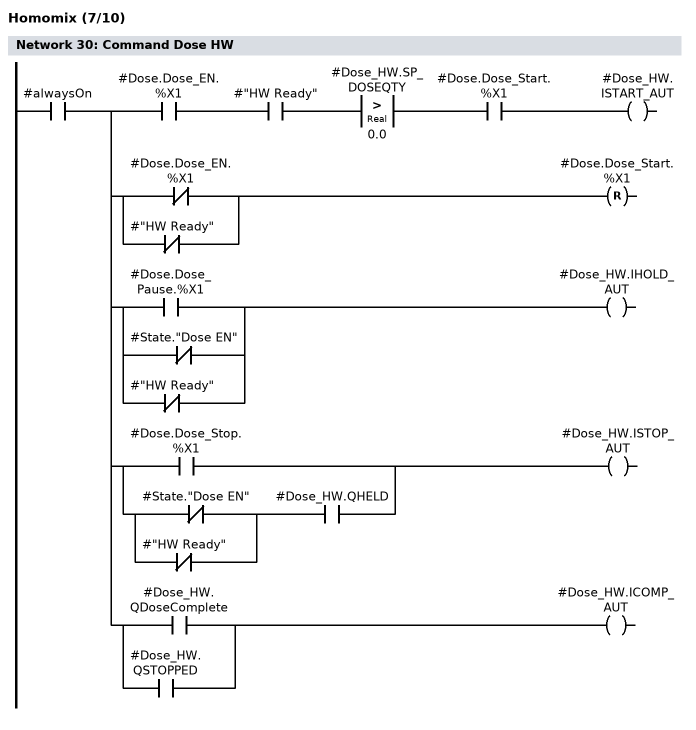
   RUNG wire#powerrail
      Contact( #alwaysOn )
      wire#w1
      Contact( #Dose.Dose_EN.%X1 )
      Contact( #"HW Ready" )
      { S7_Templates := "SrcType := Real" } GT_Contact(in1 := #Dose_HW.SP_DOSEQTY, in2 := 0.0)
      Contact( #Dose.Dose_Start.%X1 )
      Coil( #Dose_HW.ISTART_AUT )
   END_RUNG
   RUNG wire#w1
      I_Contact( #Dose.Dose_EN.%X1 )
      wire#w2
      R_Coil( #Dose.Dose_Start.%X1 )
   END_RUNG
   RUNG wire#w1
      I_Contact( #"HW Ready" )
   END_RUNG wire#w2
   RUNG wire#w1
      Contact( #Dose.Dose_Pause.%X1 )
      wire#w3
      Coil( #Dose_HW.IHOLD_AUT )
   END_RUNG
   RUNG wire#w1
      I_Contact( #State."Dose EN" )
   END_RUNG wire#w3
   RUNG wire#w1
      I_Contact( #"HW Ready" )
   END_RUNG wire#w3
   RUNG wire#w1
      Contact( #Dose.Dose_Stop.%X1 )
      wire#w4
      Coil( #Dose_HW.ISTOP_AUT )
   END_RUNG
   RUNG wire#w1
      I_Contact( #State."Dose EN" )
      wire#w5
      Contact( #Dose_HW.QHELD )
   END_RUNG wire#w4
   RUNG wire#w1
      I_Contact( #"HW Ready" )
   END_RUNG wire#w5
   RUNG wire#w1
      Contact( #Dose_HW.QDoseComplete )
      wire#w6
      Coil( #Dose_HW.ICOMP_AUT )
   END_RUNG
   RUNG wire#w1
      Contact( #Dose_HW.QSTOPPED )
   END_RUNG wire#w6
   // the same network as SCL:
   #Dose_HW.ISTART_AUT := #alwaysOn AND #Dose.Dose_EN.%X1 AND #"HW Ready" AND (#Dose_HW.SP_DOSEQTY > 0.0) AND #Dose.Dose_Start.%X1;
   IF #alwaysOn AND (NOT #Dose.Dose_EN.%X1 OR NOT #"HW Ready") THEN #Dose.Dose_Start.%X1 := FALSE; END_IF;
   #Dose_HW.IHOLD_AUT := #alwaysOn AND (#Dose.Dose_Pause.%X1 OR NOT #State."Dose EN" OR NOT #"HW Ready");
   #Dose_HW.ISTOP_AUT := #alwaysOn AND (#Dose.Dose_Stop.%X1 OR ((NOT #State."Dose EN" OR NOT #"HW Ready") AND #Dose_HW.QHELD));
   #Dose_HW.ICOMP_AUT := #alwaysOn AND (#Dose_HW.QDoseComplete OR #Dose_HW.QSTOPPED);
END_REGION

REGION Network 31: Dose HW
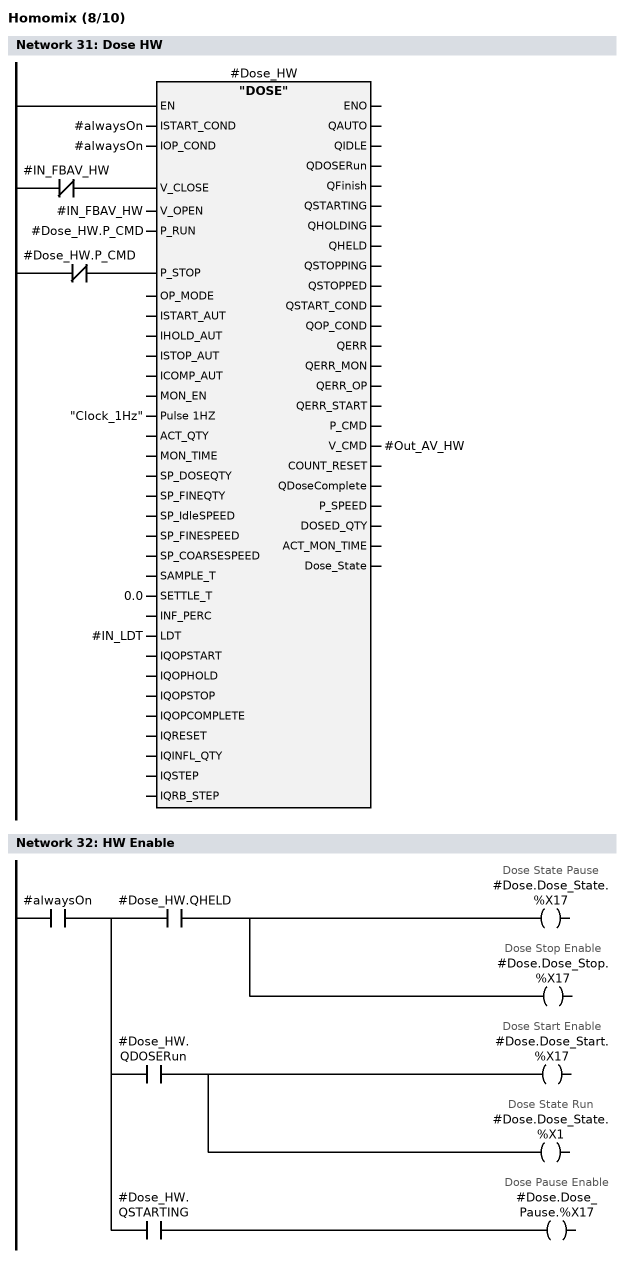
   RUNG wire#powerrail
      #Dose_HW(V_CLOSE := wire#w1, P_STOP := wire#w2, ISTART_COND := #alwaysOn, IOP_COND := #alwaysOn, V_OPEN := #IN_FBAV_HW, P_RUN := #Dose_HW.P_CMD, OP_MODE :=, ISTART_AUT :=, IHOLD_AUT :=, ISTOP_AUT :=, ICOMP_AUT :=, MON_EN :=, "Pulse 1HZ" := "Clock_1Hz", ACT_QTY :=, MON_TIME :=, SP_DOSEQTY :=, SP_FINEQTY :=, SP_IdleSPEED :=, SP_FINESPEED :=, SP_COARSESPEED :=, SAMPLE_T :=, SETTLE_T := 0.0, INF_PERC :=, LDT := #IN_LDT, IQOPSTART :=, IQOPHOLD :=, IQOPSTOP :=, IQOPCOMPLETE :=, IQRESET :=, IQINFL_QTY :=, IQSTEP :=, IQRB_STEP :=, QAUTO =>, QIDLE =>, QDOSERun =>, QFinish =>, QSTARTING =>, QHOLDING =>, QHELD =>, QSTOPPING =>, QSTOPPED =>, QSTART_COND =>, QOP_COND =>, QERR =>, QERR_MON =>, QERR_OP =>, QERR_START =>, P_CMD =>, V_CMD => #Out_AV_HW, COUNT_RESET =>, QDoseComplete =>, P_SPEED =>, DOSED_QTY =>, ACT_MON_TIME =>, Dose_State =>)
   END_RUNG
   RUNG wire#powerrail
      I_Contact( #IN_FBAV_HW )
   END_RUNG wire#w1
   RUNG wire#powerrail
      I_Contact( #Dose_HW.P_CMD )
   END_RUNG wire#w2
   // the same network as SCL:
   #Dose_HW(ISTART_COND := #alwaysOn,   // "DOSE"
            IOP_COND := #alwaysOn,
            V_CLOSE := NOT #IN_FBAV_HW,
            V_OPEN := #IN_FBAV_HW,
            P_RUN := #Dose_HW.P_CMD,
            P_STOP := NOT #Dose_HW.P_CMD,
            "Pulse 1HZ" := "Clock_1Hz",
            SETTLE_T := 0.0,
            LDT := #IN_LDT,
            V_CMD => #Out_AV_HW);
END_REGION

REGION Network 32: HW Enable
   RUNG wire#powerrail
      Contact( #alwaysOn )
      wire#w1
      Contact( #Dose_HW.QHELD )
      wire#w2
      Coil( #Dose.Dose_State.%X17 )   // Dose State Pause
   END_RUNG
   RUNG wire#w2
      Coil( #Dose.Dose_Stop.%X17 )   // Dose Stop Enable
   END_RUNG
   RUNG wire#w1
      Contact( #Dose_HW.QDOSERun )
      wire#w3
      Coil( #Dose.Dose_Start.%X17 )   // Dose Start Enable
   END_RUNG
   RUNG wire#w3
      Coil( #Dose.Dose_State.%X1 )   // Dose State Run
   END_RUNG
   RUNG wire#w1
      Contact( #Dose_HW.QSTARTING )
      Coil( #Dose.Dose_Pause.%X17 )   // Dose Pause Enable
   END_RUNG
   // the same network as SCL:
   #Dose.Dose_State.%X17 := #alwaysOn AND #Dose_HW.QHELD;   // Dose State Pause
   #Dose.Dose_Stop.%X17 := #Dose.Dose_State.%X17;   // Dose Stop Enable
   #Dose.Dose_Start.%X17 := #alwaysOn AND #Dose_HW.QDOSERun;   // Dose Start Enable
   #Dose.Dose_State.%X1 := #Dose.Dose_Start.%X17;   // Dose State Run
   #Dose.Dose_Pause.%X17 := #alwaysOn AND #Dose_HW.QSTARTING;   // Dose Pause Enable
END_REGION

REGION Network 33: HW Header Req and Valve
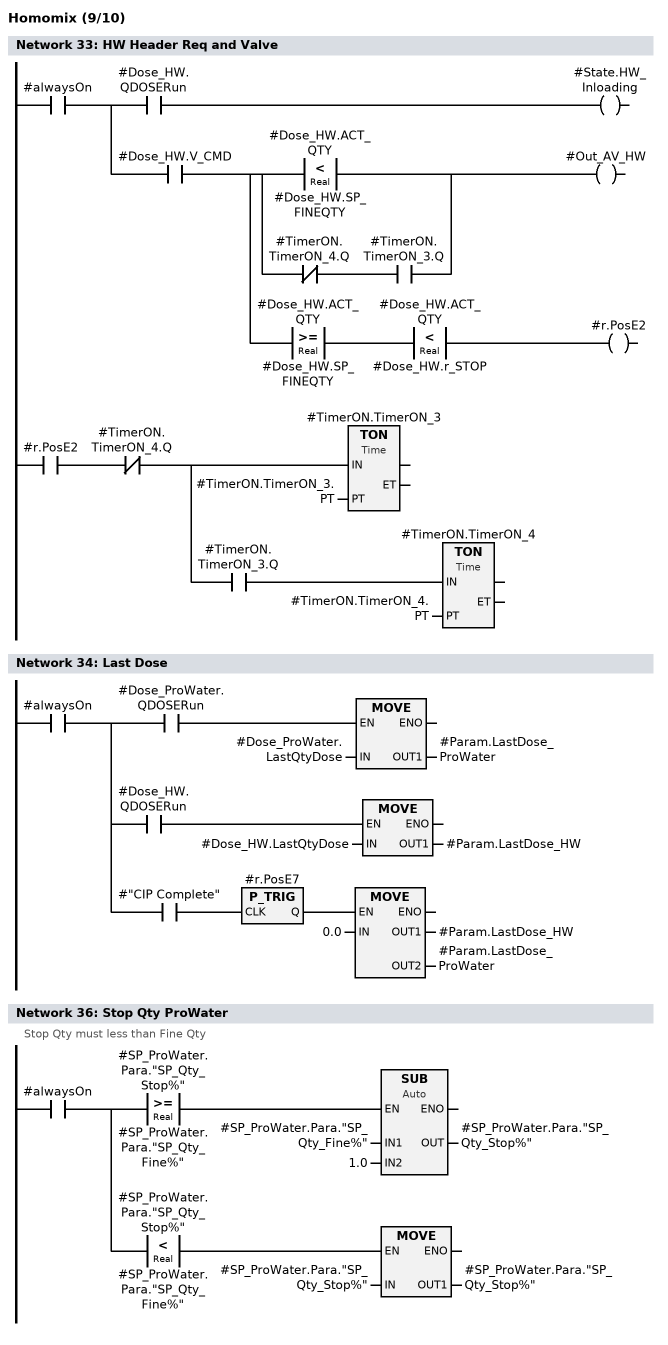
   RUNG wire#powerrail
      Contact( #alwaysOn )
      wire#w1
      Contact( #Dose_HW.QDOSERun )
      Coil( #State.HW_Inloading )
   END_RUNG
   RUNG wire#w1
      Contact( #Dose_HW.V_CMD )
      wire#w2
      { S7_Templates := "SrcType := Real" } LT_Contact(in1 := #Dose_HW.ACT_QTY, in2 := #Dose_HW.SP_FINEQTY)
      wire#w3
      Coil( #Out_AV_HW )
   END_RUNG
   RUNG wire#w2
      I_Contact( #TimerON.TimerON_4.Q )
      Contact( #TimerON.TimerON_3.Q )
   END_RUNG wire#w3
   RUNG wire#w2
      { S7_Templates := "SrcType := Real" } GE_Contact(in1 := #Dose_HW.ACT_QTY, in2 := #Dose_HW.SP_FINEQTY)
      { S7_Templates := "SrcType := Real" } LT_Contact(in1 := #Dose_HW.ACT_QTY, in2 := #Dose_HW.r_STOP)
      Coil( #r.PosE2 )
   END_RUNG
   RUNG wire#powerrail
      Contact( #r.PosE2 )
      I_Contact( #TimerON.TimerON_4.Q )
      wire#w4
      { S7_Templates := "time_type := Time" } #TimerON.TimerON_3.TON(pt := #TimerON.TimerON_3.PT, et =>)
   END_RUNG
   RUNG wire#w4
      Contact( #TimerON.TimerON_3.Q )
      { S7_Templates := "time_type := Time" } #TimerON.TimerON_4.TON(pt := #TimerON.TimerON_4.PT, et =>)
   END_RUNG
   // the same network as SCL:
   #State.HW_Inloading := #alwaysOn AND #Dose_HW.QDOSERun;
   #_w1 := #alwaysOn AND #Dose_HW.V_CMD;
   #Out_AV_HW := #_w1 AND ((#Dose_HW.ACT_QTY < #Dose_HW.SP_FINEQTY) OR (NOT #TimerON.TimerON_4.Q AND #TimerON.TimerON_3.Q));
   #r.PosE2 := #_w1 AND (#Dose_HW.ACT_QTY >= #Dose_HW.SP_FINEQTY) AND (#Dose_HW.ACT_QTY < #Dose_HW.r_STOP);
   #_w2 := #r.PosE2 AND NOT #TimerON.TimerON_4.Q;
   #TimerON.TimerON_3.TON(IN := #_w2, PT := #TimerON.TimerON_3.PT);
   #TimerON.TimerON_4.TON(IN := #_w2 AND #TimerON.TimerON_3.Q, PT := #TimerON.TimerON_4.PT);
END_REGION

REGION Network 34: Last Dose
   RUNG wire#powerrail
      Contact( #alwaysOn )
      wire#w1
      Contact( #Dose_ProWater.QDOSERun )
      Move(in := #Dose_ProWater.LastQtyDose, out1 => #Param.LastDose_ProWater)
   END_RUNG
   RUNG wire#w1
      Contact( #Dose_HW.QDOSERun )
      Move(in := #Dose_HW.LastQtyDose, out1 => #Param.LastDose_HW)
   END_RUNG
   RUNG wire#w1
      Contact( #"CIP Complete" )
      P_Trig( #r.PosE7 )
      Move(in := 0.0, out1 => #Param.LastDose_HW, out2 => #Param.LastDose_ProWater)
   END_RUNG
   // the same network as SCL:
   IF #alwaysOn AND #Dose_ProWater.QDOSERun THEN
       #Param.LastDose_ProWater := #Dose_ProWater.LastQtyDose;
   END_IF;
   IF #alwaysOn AND #Dose_HW.QDOSERun THEN #Param.LastDose_HW := #Dose_HW.LastQtyDose; END_IF;
   #_w1 := #alwaysOn AND #"CIP Complete";
   #_w2 := #_w1 AND NOT #r.PosE7;   // rising edge
   #r.PosE7 := #_w1;
   IF #_w2 THEN
       #Param.LastDose_HW := 0.0;
       #Param.LastDose_ProWater := 0.0;
   END_IF;
END_REGION

REGION Network 36: Stop Qty ProWater
   // Stop Qty must less than Fine Qty
   RUNG wire#powerrail
      Contact( #alwaysOn )
      wire#w1
      { S7_Templates := "SrcType := Real" } GE_Contact(in1 := #SP_ProWater.Para."SP_Qty_Stop%", in2 := #SP_ProWater.Para."SP_Qty_Fine%")
      Sub(in1 := #SP_ProWater.Para."SP_Qty_Fine%", in2 := 1.0, out => #SP_ProWater.Para."SP_Qty_Stop%")
   END_RUNG
   RUNG wire#w1
      { S7_Templates := "SrcType := Real" } LT_Contact(in1 := #SP_ProWater.Para."SP_Qty_Stop%", in2 := #SP_ProWater.Para."SP_Qty_Fine%")
      Move(in := #SP_ProWater.Para."SP_Qty_Stop%", out1 => #SP_ProWater.Para."SP_Qty_Stop%")
   END_RUNG
   // the same network as SCL:
   IF #alwaysOn AND (#SP_ProWater.Para."SP_Qty_Stop%" >= #SP_ProWater.Para."SP_Qty_Fine%") THEN
       #SP_ProWater.Para."SP_Qty_Stop%" := #SP_ProWater.Para."SP_Qty_Fine%" - 1.0;
   END_IF;
   IF #alwaysOn AND (#SP_ProWater.Para."SP_Qty_Stop%" < #SP_ProWater.Para."SP_Qty_Fine%") THEN
       #SP_ProWater.Para."SP_Qty_Stop%" := #SP_ProWater.Para."SP_Qty_Stop%";
   END_IF;
END_REGION

REGION Network 37: Stop Qty HW
   // Stop Qty must less than Fine Qty
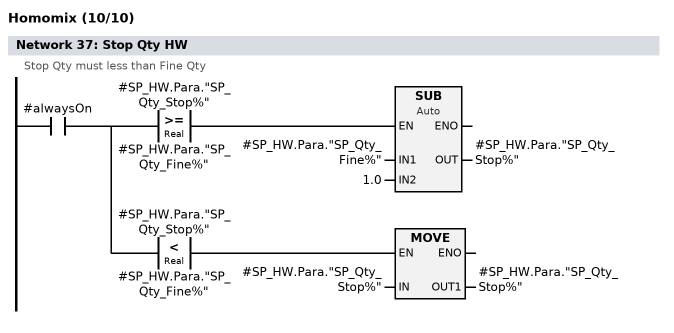
   RUNG wire#powerrail
      Contact( #alwaysOn )
      wire#w1
      { S7_Templates := "SrcType := Real" } GE_Contact(in1 := #SP_HW.Para."SP_Qty_Stop%", in2 := #SP_HW.Para."SP_Qty_Fine%")
      Sub(in1 := #SP_HW.Para."SP_Qty_Fine%", in2 := 1.0, out => #SP_HW.Para."SP_Qty_Stop%")
   END_RUNG
   RUNG wire#w1
      { S7_Templates := "SrcType := Real" } LT_Contact(in1 := #SP_HW.Para."SP_Qty_Stop%", in2 := #SP_HW.Para."SP_Qty_Fine%")
      Move(in := #SP_HW.Para."SP_Qty_Stop%", out1 => #SP_HW.Para."SP_Qty_Stop%")
   END_RUNG
   // the same network as SCL:
   IF #alwaysOn AND (#SP_HW.Para."SP_Qty_Stop%" >= #SP_HW.Para."SP_Qty_Fine%") THEN
       #SP_HW.Para."SP_Qty_Stop%" := #SP_HW.Para."SP_Qty_Fine%" - 1.0;
   END_IF;
   IF #alwaysOn AND (#SP_HW.Para."SP_Qty_Stop%" < #SP_HW.Para."SP_Qty_Fine%") THEN
       #SP_HW.Para."SP_Qty_Stop%" := #SP_HW.Para."SP_Qty_Stop%";
   END_IF;
END_REGION
END_FUNCTION_BLOCK
